Fanuc KAREL source: kt00535.KL

-- PROVISIONAL review KL for V1013-1; original PC SHA256 54a33fdd11073c4e07d33206fd9614d7038b19ab342306de294865b34f802a22
-- Incomplete behavior may be omitted. Consult companion uncertainty JSON. Do not deploy.
PROGRAM KT00535
%NOLOCKGROUP
-- UNRESOLVED_DECL P1 type=000199
-- UNRESOLVED_DECL P2 type=000101
-- UNRESOLVED_DECL OUT type=000102
BEGIN
  -- UNRESOLVED_PC offsets 5-39; opcodes 49,7E,49,60,7E,4A
  -- UNRESOLVED_PC offsets 44-48; opcodes 7F
END KT00535
